PROGRAM P_Demo_FB_HVACScaleXX
VAR
    fb : FB_HVACScaleXX;                            // 被演示 FB 实例
    lrX_in : LREAL := 0.0;
    lrX0n_in : LREAL := 0.0;
    lrY0n_in : LREAL := 0.0;
    bLmt_in : BOOL := FALSE;
    lrY_out : LREAL;
    bError_out : BOOL;
    eErrorCode_out : E_HVACErrorCodes;
    udiErrorArgument_out : UDINT;
END_VAR

// ============================================================================
// Tc2_HVAC.FB_HVACScaleXX 演示程序
// ============================================================================
// 场景：把本 FB 实例化到一个 PLC 程序里，每周期单次调用；按需要把 VAR_INPUT 与
//       VAR_IN_OUT 接到工程信号；VAR_OUTPUT 写入对应监视变量。
// 价值：使用本 FB 比手写状态机 / 控制算法节省大量代码；与 Tc2_HVAC 体系内其它 FB
//       直接对接，命名 / 持久化 / 模式仲裁等约定一致。具体语义见 FB_HVACScaleXX.md 主文档。
// 验证步骤：
//   1. 右键 PLC 项目下 POUs 文件夹 → Add → Existing Item → 选本 .TcPOU 文件
//   2. 引用 Tc2_HVAC（References → Add library）
//   3. 编译 → 登录 → 运行
//   4. 在线写各 *_in 输入信号触发 FB；在线 monitor *_out 引脚观察状态
// ============================================================================

fb(
    lrX := lrX_in,
    lrX0n := lrX0n_in,
    lrY0n := lrY0n_in,
    bLmt := bLmt_in,
    lrY => lrY_out,
    bError => bError_out,
    eErrorCode => eErrorCode_out,
    udiErrorArgument => udiErrorArgument_out
);

END_PROGRAM

(* stored: Version 1.1.0.1, ProductVersion 3.1.4024.5
   POU P_Demo_FB_HVACScaleXX: Id {50903709-5144-5adc-b94f-f0afe8a15cf7}, SpecialFunc None *)
